(* IEC 61131-3 sources: plc_projects/rasi_feed_batching_2/Scripts_cursor/review_output/st_export (part 4) *)

    31:
        IF Semi_Has_Active_Bins THEN
            Active_Material_ID := 0;
            Active_Bin_ID := 0;
            Active_Target_Weight := 0.0;
            Active_Live_Weight := 0.0;
            GVL.Semi_Auto_Active_Target_Weight := 0.0;
            GVL.Semi_Auto_Active_Live_Weight := 0.0;
            Excess_Alarm := FALSE;
            GVL.Semi_Auto_Excess_Alarm := FALSE;
            FOR i := 1 TO 10 DO
                Semi_Auto_Bin[i] := FALSE;
                semi_auto_bin_cutoff[i] := FALSE;
                semi_auto_bin_motor[i] := FALSE;
            END_FOR;
            Status_Message := 'Semi-Auto [Step 31]: Settling Delay in progress...';
            IF Settle_Phase = 0 THEN
                Completion_Timer(IN := FALSE);
                Settle_Phase := 1;
            ELSE
                Completion_Timer(IN := TRUE, PT := Effective_Delay);
                IF Completion_Timer.Q THEN
                    Completion_Timer(IN := FALSE);
                    Settle_Phase := 0;
                    Current_Step := 32;
                END_IF;
            END_IF;
        ELSE
            Current_Step := 32;
        END_IF;

    32:
        Active_Material_ID := 0;
        Active_Bin_ID := 0;
        Excess_Alarm := FALSE;
        Sequence_Complete := TRUE;
        GVL.Semi_Auto_Sequence_Complete := TRUE;
        IF NOT GVL.Auto_Sequence_Complete THEN
            Status_Message := 'Semi-Auto [Step 32]: Semi done — waiting for Auto to finish';
        ELSIF (Cycle_Manager_State = 5) OR Between_Cycle_Hold THEN
            Status_Message := 'Semi-Auto [Step 32]: Cycle done — empty BOTH scales then Next_Cycle_Start';
        ELSIF (GVL.Target_Batch_Cycles > 1) AND (GVL.Completed_Batch_Cycles >= 1)
            AND (GVL.Completed_Batch_Cycles < GVL.Target_Batch_Cycles) THEN
            Status_Message := 'Semi-Auto [Step 32]: Both done — waiting State 5 / Next_Cycle_Start';
        ELSIF (GVL.Current_Batch_Cycle >= GVL.Target_Batch_Cycles) AND (GVL.Target_Batch_Cycles > 0) THEN
            Status_Message := 'Semi-Auto [Step 32]: All target batch cycles complete';
        ELSE
            Status_Message := 'Semi-Auto [Step 32]: Cycle sequences complete';
        END_IF;
END_CASE;

Last_Step := Current_Step;

(* Synchronize physical output arrays to GVL *)
FOR i := 1 TO 10 DO
    GVL.Semi_Auto_Bin[i] := Semi_Auto_Bin[i];
    GVL.semi_auto_bin_cutoff[i] := semi_auto_bin_cutoff[i];
    GVL.semi_auto_bin_motor[i] := semi_auto_bin_motor[i];
END_FOR;

(* Synchronize live cycle progress to outputs *)
Semi_Auto_Current_Batch_Cycle := GVL.Current_Batch_Cycle;
Semi_Auto_Completed_Batch_Cycles := GVL.Completed_Batch_Cycles;
Semi_Auto_All_Cycles_Complete := GVL.All_Cycles_Complete;

(* When cycle handshake done, show Step32 not last dosing step on HMI *)
IF Sequence_Complete AND (Current_Step >= 1) AND (Current_Step <= 10) THEN
    Current_Step := 32;
END_IF;
GVL.Semi_Auto_Current_Step := Current_Step;
(* HMI Active Mat/Bin: only while dosing steps 1..10 with valid live mapping *)
(* During inter-bin settle keep Settle_Hold_* for TRUE and FALSE — do not overwrite with next bin *)
IF Inter_Bin_Settling AND (Settle_Hold_Step >= 1) THEN
    Active_Material_ID := Settle_Hold_Mat;
    Active_Bin_ID := Settle_Hold_Step;
    Active_Target_Weight := Settle_Hold_Target;
    actual_bin := load_cell_value - bin_last_weight;
    IF actual_bin < 0.0 THEN
        actual_bin := 0.0;
    END_IF;
    Actual_Weights[Settle_Hold_Step] := actual_bin;
    Active_Live_Weight := actual_bin;
    GVL.Semi_Auto_Current_Step := Settle_Hold_Step;
ELSIF (Current_Step >= 1) AND (Current_Step <= 10) AND (NOT Inter_Bin_Settling) THEN
    Mat_Idx := Semi_Auto_Bin_Material_Mapping[Current_Step];
    target_weight := 0.0;
    IF (Mat_Idx >= 1) AND (Mat_Idx <= 20) THEN
        target_weight := GVL.Recipe_Weights[Mat_Idx];
    END_IF;
    IF (target_weight <= 0.0) AND (PersistentVars.Ret_Semi_Bin_Target_Weights[Current_Step] > 0.0) THEN
        target_weight := PersistentVars.Ret_Semi_Bin_Target_Weights[Current_Step];
        IF (Mat_Idx < 1) OR (Mat_Idx > 20) THEN
            IF PersistentVars.Ret_Semi_Bin_Target_Weights[Current_Step] > 0.0 THEN
                Mat_Idx := PersistentVars.Ret_Semi_Bin_Material_Mapping[Current_Step];
            ELSE
                Mat_Idx := 0;
            END_IF;
        END_IF;
    END_IF;
    IF (Mat_Idx < 1) OR (Mat_Idx > 20) OR (target_weight <= 0.0) THEN
        Active_Material_ID := 0;
        Active_Bin_ID := 0;
        Active_Target_Weight := 0.0;
        Active_Live_Weight := 0.0;
    ELSE
        (* Dosing: keep Actual_Weights in sync with live scale (excess / tailings) *)
        actual_bin := load_cell_value - bin_last_weight;
        IF actual_bin < 0.0 THEN
            actual_bin := 0.0;
        END_IF;
        Actual_Weights[Current_Step] := actual_bin;
        Active_Live_Weight := actual_bin;
    END_IF;
ELSE
    Active_Material_ID := 0;
    Active_Bin_ID := 0;
    Active_Target_Weight := 0.0;
    Active_Live_Weight := 0.0;
END_IF;
GVL.Semi_Auto_Active_Mat := Active_Material_ID;
GVL.Semi_Auto_Active_Bin := Active_Bin_ID;
GVL.Semi_Auto_Active_Target_Weight := Active_Target_Weight;
GVL.Semi_Auto_Active_Live_Weight := Active_Live_Weight;
(* Mirror Actual_Weights to HMI every scan — dosing, excess, inter-bin tailings *)
Semi_Auto_Sum_ActWeight := 0.0;
FOR i := 1 TO 10 DO
    GVL.Semi_Auto_Weights[i] := Actual_Weights[i];
    Semi_Auto_Sum_ActWeight := Semi_Auto_Sum_ActWeight + Actual_Weights[i];
END_FOR;
GVL.Semi_Auto_Total_Actual_Weight := Semi_Auto_Sum_ActWeight;
(* Per-bin target setpoints — bin index 1..10; mirror to GVL.Semi_Auto_Target_Weights (plant %MD410) *)
(* Do not zero on CMS4 / All_Cycles_Complete (Auto holds recipe targets after last cycle) *)
IF (Cycle_Manager_State = 0) AND (NOT GVL.Run) AND (NOT PersistentVars.Ret_Semi_Process_Was_Active)
    AND (NOT GVL.All_Cycles_Complete) AND (Cycle_Manager_State <> 4) THEN
    FOR i := 1 TO 10 DO
        Semi_Auto_Target_Weight[i] := 0.0;
        GVL.Semi_Auto_Target_Weights[i] := 0.0;
    END_FOR;
ELSE
    FOR i := 1 TO 10 DO
        Mat_Idx := Semi_Auto_Bin_Material_Mapping[i];
        IF (Mat_Idx < 1) OR (Mat_Idx > 20) THEN
            IF PersistentVars.Ret_Semi_Bin_Target_Weights[i] > 0.0 THEN
                Mat_Idx := PersistentVars.Ret_Semi_Bin_Material_Mapping[i];
            ELSE
                Mat_Idx := 0;
            END_IF;
        END_IF;
        target_weight := 0.0;
        IF (Mat_Idx >= 1) AND (Mat_Idx <= 20) THEN
            target_weight := GVL.Recipe_Weights[Mat_Idx];
        END_IF;
        IF (target_weight <= 0.0) AND (PersistentVars.Ret_Semi_Bin_Target_Weights[i] > 0.0) THEN
            target_weight := PersistentVars.Ret_Semi_Bin_Target_Weights[i];
        END_IF;
        Semi_Auto_Target_Weight[i] := target_weight;
        GVL.Semi_Auto_Target_Weights[i] := target_weight;
    END_FOR;
END_IF;
(* Semi snapshot: only clear retain when all cycles finished (CMS4). Never clear on Run=FALSE power loss. *)
IF Cycle_Manager_State = 4 THEN
    PersistentVars.Ret_Semi_Process_Was_Active := FALSE;
    PersistentVars.Ret_Semi_GVL_Run := FALSE;
    PersistentVars.Ret_Semi_Cycle_Manager_State := 0;
    PersistentVars.Ret_Semi_Current_Step := 0;
    PersistentVars.Ret_Semi_Between_Cycle_Hold := FALSE;
    PersistentVars.Ret_Semi_Active_Material_ID := 0;
    PersistentVars.Ret_Semi_Active_Bin_ID := 0;
    PersistentVars.Ret_Semi_Active_Target_Weight := 0.0;
    PersistentVars.Ret_Semi_Active_Live_Weight := 0.0;
    PersistentVars.Ret_Semi_Resume_Step := 0;
ELSIF (GVL.Run OR (Cycle_Manager_State = 1) OR (Cycle_Manager_State = 5) OR Between_Cycle_Hold) AND (Cycle_Manager_State <> 4) THEN
    j := 0;
    FOR i := 1 TO 10 DO
        Mat_Idx := Semi_Auto_Bin_Material_Mapping[i];
        IF (Mat_Idx < 1) OR (Mat_Idx > 20) THEN
            IF PersistentVars.Ret_Semi_Bin_Target_Weights[i] > 0.0 THEN
                Mat_Idx := PersistentVars.Ret_Semi_Bin_Material_Mapping[i];
            ELSE
                Mat_Idx := 0;
            END_IF;
        END_IF;
        target_weight := 0.0;
        IF (Mat_Idx >= 1) AND (Mat_Idx <= 20) THEN
            target_weight := GVL.Recipe_Weights[Mat_Idx];
        END_IF;
        IF (target_weight <= 0.0) AND (PersistentVars.Ret_Semi_Bin_Target_Weights[i] > 0.0) THEN
            target_weight := PersistentVars.Ret_Semi_Bin_Target_Weights[i];
        END_IF;
        IF (Mat_Idx >= 1) AND (Mat_Idx <= 20) AND (target_weight > 0.0) THEN
            IF Actual_Weights[i] < (target_weight - 0.05) THEN
                j := i;
                EXIT;
            END_IF;
        END_IF;
    END_FOR;
    IF (j > 0) AND ((Cycle_Manager_State = 5) OR (Current_Step >= 31) OR Between_Cycle_Hold) THEN
        PersistentVars.Ret_Semi_Process_Was_Active := TRUE;
        PersistentVars.Ret_Semi_Current_Step := j;
        PersistentVars.Ret_Semi_Cycle_Manager_State := 1;
        PersistentVars.Ret_Semi_Between_Cycle_Hold := FALSE;
        PersistentVars.Ret_Semi_Resume_Step := j;
    ELSE
        PersistentVars.Ret_Semi_Process_Was_Active := TRUE;
        PersistentVars.Ret_Semi_Current_Step := Current_Step;
        PersistentVars.Ret_Semi_Cycle_Manager_State := Cycle_Manager_State;
        PersistentVars.Ret_Semi_Between_Cycle_Hold := Between_Cycle_Hold;
        PersistentVars.Ret_Semi_Last_Batch_Cycle := Last_Batch_Cycle;
        IF (Cycle_Manager_State = 1) AND (Current_Step >= 1) AND (Current_Step <= 10) THEN
            PersistentVars.Ret_Semi_Resume_Step := Current_Step;
        ELSIF (Cycle_Manager_State = 5) OR (Cycle_Manager_State = 4) OR (Current_Step >= 31) THEN
            PersistentVars.Ret_Semi_Resume_Step := 0;
        END_IF;
    END_IF;
    PersistentVars.Ret_Semi_bin_last_weight := bin_last_weight;
    PersistentVars.Ret_Semi_GVL_Run := GVL.Run;
    PersistentVars.Ret_Semi_Current_Batch_Cycle := GVL.Current_Batch_Cycle;
    PersistentVars.Ret_Semi_Completed_Batch_Cycles := GVL.Completed_Batch_Cycles;
    PersistentVars.Ret_Semi_Target_Batch_Cycles := GVL.Target_Batch_Cycles;
    PersistentVars.Ret_Semi_Active_Material_ID := Active_Material_ID;
    PersistentVars.Ret_Semi_Active_Bin_ID := Active_Bin_ID;
    PersistentVars.Ret_Semi_Active_Target_Weight := Active_Target_Weight;
    PersistentVars.Ret_Semi_Active_Live_Weight := Active_Live_Weight;
    FOR i := 1 TO 10 DO
        PersistentVars.Ret_Semi_Actual_Weights[i] := Actual_Weights[i];
        Mat_Idx := Semi_Auto_Bin_Material_Mapping[i];
        IF (Mat_Idx < 1) OR (Mat_Idx > 20) THEN
            IF PersistentVars.Ret_Semi_Bin_Target_Weights[i] > 0.0 THEN
                Mat_Idx := PersistentVars.Ret_Semi_Bin_Material_Mapping[i];
            ELSE
                Mat_Idx := 0;
            END_IF;
        END_IF;
        IF (Mat_Idx >= 1) AND (Mat_Idx <= 20) THEN
            PersistentVars.Ret_Semi_Bin_Material_Mapping[i] := Mat_Idx;
            IF GVL.Recipe_Weights[Mat_Idx] > 0.0 THEN
                PersistentVars.Ret_Semi_Bin_Target_Weights[i] := GVL.Recipe_Weights[Mat_Idx];
            END_IF;
        END_IF;
    END_FOR;
END_IF;

(* Drop any tare request if scales not empty (batch still on scale after cycle complete) *)
IF NOT Scale_Empty_OK THEN
    Tare_Pulse_Req := FALSE;
END_IF;

(* TARE PULSE — end of scan (after sequence / Next_Cycle set Tare_Pulse_Req); BOTH scales LT limit *)
IF Tare_Pulse_Req THEN
    IF Scale_Empty_OK THEN
        Tare_Semi_Auto_Batch := TRUE;
        Status_Message := 'Semi-Auto [Tare]: Scales empty - Tare_Semi_Auto_Batch pulse';
    ELSE
        Tare_Semi_Auto_Batch := FALSE;
        Status_Message := CONCAT('Semi-Auto [Tare blocked]: Scale >= ', CONCAT(REAL_TO_STRING(eff_empty_limit), ' kg — dump batch first'));
    END_IF;
    Tare_Pulse_Req := FALSE;
END_IF;

(* Hard interlock: never Tare when live load >= Empty_Weight_Limit (either scale) *)
IF NOT Scale_Empty_OK THEN
    Tare_Semi_Auto_Batch := FALSE;
END_IF;

(* ---- batching14.st ---- *)
(* POU: batching14 *)

=== DECLARATION ===
PROGRAM batching14
VAR
	Auto_Ctrl: Auto_Batching_V15;
	Semi_Auto_Ctrl: Semi_Auto_Batching_V15;
	Auto_Complete: BOOL;
	Semi_Auto_Complete: BOOL;
	Auto_Err: INT;
	Auto_Msg: STRING;
	Semi_Auto_Err: INT;
	Semi_Auto_Msg: STRING;
	AutoBatchScale: MODRTUMAST;
	ModEnabler: BLINK;
	SamyakRaw: ARRAY[0..1] OF DINT;
	AutBatchRaw: ARRAY[0..1] OF DINT;
	SemAutoScale: MODRTUMAST;
	SemiAutoScaleRaw: ARRAY[0..1] OF DINT;
	AutoBatchSamyak: REAL;
	FB_Samyak_Multi_1: FB_Samyak_Multi;
	FB_Samyak_Control_1: FB_Samyak_Control;
	Run_PB_1: BOOL;
	Next_Cycle_Start: BOOL;
	TP_1: TP;
	TP_ON: BOOL;
	TP_Out: BOOL;
	TP_Et: TIME;
	arrTare_Cmds: ARRAY[1..4] OF BOOL;
END_VAR

=== IMPLEMENTATION ===
(* empty textual body - see batching14_fbd.xml for FBD *)
